Fanuc KAREL source: TAN.kl

PROGRAM T
%NOLOCKGROUP
VAR
 v0 : REAL
 res : REAL
BEGIN
 res = TAN(v0)
END T
